// TwinCAT 3 PLC project PLC1
// ProgramVersion: 3.1.4023.0
// libraries:
//   Tc2_MC2, * (Beckhoff Automation GmbH)
//   Tc2_Standard, * (Beckhoff Automation GmbH)
//   Tc2_System, * (Beckhoff Automation GmbH)
//   Tc3_Module, * (Beckhoff Automation GmbH)
//   Tc3_XPlanarStandard, * (Beckhoff Automation GmbH)
//   XboxControllerUtilities, * (Beckhoff Community)
// project tree:
//   / PlcTask.TcTTO
//   POUs/ MAIN.TcPOU
// real-time tasks:
//   TASK XPlanar Task3: cycle T#250us, priority 1, ADS port 350
//   TASK Job Task: cycle default, priority 32
//   TASK MC-Task (MET): cycle T#2ms, priority 3, ADS port 521
//   TASK MC-Task (MPT): cycle T#10ms, priority 8, ADS port 531
//   TASK PlcTask: cycle T#10ms, priority 20, ADS port 351
// variable links:
//   TcCOM Objects/XPlanar/Mover4330_1 <-> XPlanar MC Project/Axes/Mover4330_1
//     InputsFromNC3/NC3ToHW <-> McToIo/STD
//     OutputsToNC3/HWToNC3 <-> IoToMc/STD
//   PLC1 Instance <-> XPlanar MC Project/Axes/Mover4330_1
//     PlcTask Inputs/MAIN.XPlanarMover.stMoverRef.MCTOPLC/ACT <-> McToPlc/ACT
//     PlcTask Inputs/MAIN.XPlanarMover.stMoverRef.MCTOPLC/COORDMODE <-> McToPlc/COORDMODE
//     PlcTask Inputs/MAIN.XPlanarMover.stMoverRef.MCTOPLC/SET <-> McToPlc/SET
//     PlcTask Inputs/MAIN.XPlanarMover.stMoverRef.MCTOPLC/SETONTRACK <-> McToPlc/SETONTRACK
//     PlcTask Inputs/MAIN.XPlanarMover.stMoverRef.MCTOPLC/STD <-> McToPlc/STD
//     PlcTask Outputs/MAIN.XPlanarMover.stMoverRef.PLCTOMC/STD <-> PlcToMc/STD

CONFIGURATION PLC1
    RESOURCE PLC ON TwinCAT3
        TASK PlcTask(INTERVAL := T#10ms, PRIORITY := 20);
        PROGRAM MAIN WITH PlcTask : MAIN;
    END_RESOURCE
END_CONFIGURATION

// ---- POUs/MAIN.TcPOU
PROGRAM MAIN
VAR
	XboxController				: FB_Xbox_Controller('',1);
	
	XPlanarMover				: FB_XPlanarMoverStandard;
	bEnableMover				: BOOL := TRUE;

	
	fbXbox_2D_Joystick_XPlanar	: FB_Xbox_2D_Joystick_XPlanar;
	stOptions					: ST_Xbox_2D_Joystick_XPlanar_Options;
	bEnableJog					: BOOL;
	eJogMode					: E_Xbox_XPlanar_JogMode;
END_VAR

XPlanarMover.Cycle();
XboxController.Cycle();

IF bEnableMover THEN
	XPlanarMover.Enable(slogMessage := 'Enabling Mover');
	IF XPlanarMover.P_Enable.Done THEN
		bEnableMover := FALSE;
	END_IF
END_IF


stOptions.eJog_Mode 		:= eJogMode;
stOptions.fFastJog_Trigger 	:= XboxController.P_Left_Trigger;
stOptions.bFastJog_Button	:= XboxController.P_Buttons.bA_Button;

fbXbox_2D_Joystick_XPlanar.Jog(
								bEnable:= bEnableJog AND XboxController.P_Status.bConnected, 
								stJoystick:= XboxController.P_Left_Joystick, 
								xpMover:= XPlanarMover, 
								stOptions:= stOptions);

END_PROGRAM
